// TIA Portal V20 export
// export: Created 2025-12-01T14:57:23.2203622Z, ExportSetting None, DisplayName Totally Integrated Automation Portal, DisplayVersion V20 Update 3, DisplayName TIA Portal Openness, DisplayVersion V20 Update 3, DisplayName TIA Portal Version Control Interface, DisplayVersion V20 Update 3, DisplayName STEP 7 Professional, DisplayVersion V20 Update 3, DisplayName STEP 7 Safety, DisplayVersion V20 Update 2, DisplayName WinCC Basic/Comfort/Advanced, DisplayVersion V20 Update 3, DisplayName WinCC Professional, DisplayVersion V20 Update 3, DisplayName WinCC Unified, DisplayVersion V20 Update 3
DATA_BLOCK "DB851_SalidaMesaMultiplesDestinos"   // DB851
{ S7_Optimized_Access := 'FALSE' }
AUTHOR : TRACKING
NAME : 20141014
VERSION : 4.0
// stored: AutoNumber false
   VAR
      MesaSalida : Array[0..30] of Struct   // Variable provisional
         Origen : UInt;
         Destino : UInt;
         Intermedia : UInt;
      END_STRUCT;
   END_VAR
BEGIN
END_DATA_BLOCK
